FUNCTION SinusFunction : REAL
VAR_INPUT
	A : 	REAL; 		//Amplitude
	yoff : 	REAL;		//Offset
	w : 	REAL;		//Kreisfrequenz
	t : 	REAL;		//Zeit
END_VAR
VAR
END_VAR

SinusFunction := A * sin(w*t) + yoff;
RETURN;

END_FUNCTION

(* stored: Version 1.1.0.1, ProductVersion 3.1.4024.13
   POU SinusFunction: Id {ea880a9a-fb9c-4955-a99d-c49b67123bd6}, SpecialFunc None *)
